FUNCTION_BLOCK HydraulicCylinder
VAR_INPUT
	PressureBoreSide: LREAL;
	PressureRodSide: LREAL;
	param : ST_pValveControlledCylinder;
END_VAR
VAR_OUTPUT
	PistonAcceleration: LREAL;
	PistonVelocity : LREAL;
	PistonPosition : LREAL;
	Aa: LREAL;
	Ab: LREAL;
END_VAR
VAR
	ssMethodType : SINT := 1; 
	fbPistonVelocity : DiscreteTimeIntegrator_Init;
	fbPistonPosition : DiscreteTimeIntegrator_Init;
	Ffric : LREAL;
	Fhyd : LREAL;

END_VAR


(* Outputs for Atomic SubSystem: '<Root>/HydraulicCylinder' *)
(* Outport: '<Root>/PistonAcceleration' incorporates:
 *  Gain: '<S1>/Gain1'
 *  Gain: '<S1>/Gain2'
 *  Product: '<S1>/Divide '
 *  Product: '<S1>/Product'
 *  Product: '<S1>/Product1'
 *  Sum: '<S1>/sum' *)
 
//Area Cylinder
Aa := EXPT(param.DBore,2) * (param.pi/4.0);
Ab := (EXPT(param.DBore,2) - EXPT(param.DRod,2)) * (param.pi/4.0);

Fhyd := PressureBoreSide * Aa - PressureRodSide * Ab;
Ffric := param.FrictionConstant*PistonVelocity;
 
PistonAcceleration := (Fhyd - Ffric - param.ExternalForce) / param.EffectiveMass;
(* End of Outputs for SubSystem: '<Root>/HydraulicCylinder' *)

fbPistonVelocity(
	ssMethodType := ssMethodType,
	tCycle := param.tCycle,
	In := PistonAcceleration,
	Init := param.v0,
	minOut := -param.vMax,
	maxOut := param.vMax,
	Out => PistonVelocity
	);
	
fbPistonPosition(
	ssMethodType := ssMethodType,
	tCycle := param.tCycle,
	In := PistonVelocity,
	Init := param.x0,
	minOut := 0,
	maxOut := param.xMax,
	Out => PistonPosition
	);

//IF PistonPosition >= param.xMax THEN 
//	PistonPosition := param.xMax;
//ELSIF PistonPosition <= 0 THEN 
//	PistonPosition := 0;
//END_IF;

END_FUNCTION_BLOCK

(* stored: Version 1.1.0.1, ProductVersion 3.1.4024.9
   POU HydraulicCylinder: Id {3bf06456-7c7d-48f2-a9cc-e4b64f4dae07}, SpecialFunc None *)
